KUKA KRL data list: select.dat

&ACCESS RV
&REL 182
&PARAM TPVW_VERSION = 8.1.8
DEFDAT  SELECT
INT T_NR=0
ENDDAT
